(* IEC 61131-3 sources: ax-lightloop/src, 7 files *)

(* ---- LedStructs.st ---- *)
TYPE
    ///LedHw relative struct for IO assignment
    LedHw : STRUCT
        Red AT %X0.0 : BOOL;
        Yellow AT %X0.1 : BOOL;
        Green AT %X0.2 : BOOL;
    END_STRUCT;
END_TYPE

TYPE
    ///Leds array for passing bools
    Leds : STRUCT
        Red  : BOOL;
        Yellow  : BOOL;
        Green  : BOOL;
    END_STRUCT;
END_TYPE

(* ---- ILed.st ---- *)
/// Iled interface, every LED class should atleast have these functions
INTERFACE ILed
    /// GetState
    /// Method to get the state
    /// Return value: BOOL
    METHOD GetState : BOOL
    END_METHOD
    /// TurnOn
    /// Method to turn ON the LED
    /// Return value: BOOL
    METHOD TurnOn
    END_METHOD
    /// TurnOff
    /// Method to turn OFF the LED
    /// Return value: BOOL
    METHOD TurnOff
    END_METHOD

END_INTERFACE

(* ---- ITrafficLight.st ---- *)
INTERFACE ITrafficlight //ITrafficlight interfaces defines the minimum requirements for a lightstack

    /// GetState
    /// Method to get the current state of the TrafficLight
    /// Return value: state int
    METHOD GetState : int
    END_METHOD
    /// GetLedEquipmentState
    /// Method to get the current state of the Led's
    /// Return value: redHw :BOOL; yellowHw :BOOL; greenHw :BOOL;
    METHOD GetLedEquipmentState
        VAR_OUTPUT
            Leds: leds;
        END_VAR
        END_METHOD
    /// Go
    /// Method set the current state of the TrafficLight to Go
    /// Return value: success bool
    METHOD Go : BOOL
    END_METHOD
    /// Stop
    /// Method set the current state of the TrafficLight to Stop
    /// Return value: success bool
    METHOD Stop : BOOL
    END_METHOD
    /// Flash
    /// Method set the current state of the TrafficLight to Flash for idlemode
    /// Return value: none
    METHOD Flash
    END_METHOD
    /// Stop
    /// Method set the current state of the TrafficLight to Idle
    /// Return value: none
    METHOD  SetIdleMode
        VAR_INPUT
            Set : BOOL;
        END_VAR
    END_METHOD
END_INTERFACE

(* ---- led.st ---- *)
CLASS Led IMPLEMENTS Iled //This Class implements the Iled interface, to make sure it complies
    VAR PRIVATE //Private VAR section, only accesible from inside this class
        IsOn : BOOL; //Private BOOl to keep track of the LED state
    END_VAR
    ///This overwrites the comment defined in the interface
    METHOD PUBLIC GetState : BOOL
        GetState := IsOn; //Get the private state BOOL
        ;
    END_METHOD

    METHOD PUBLIC TurnOn
        IsOn := TRUE; //Set the state to ON
        ;
    END_METHOD

    METHOD PUBLIC TurnOff
        IsOn := FALSE; //Set the state to OFF
        ;
    END_METHOD

    /// Toggle
    /// This Method will Toggle the LED, this is not defined in the interface
    /// Return value: BOOL
    METHOD PUBLIC Toggle
        IF IsOn THEN //If the LED IsOn = true then set the LED to OFF
            IsOn := FALSE;
        ELSE
            IsOn := TRUE; //If the LED IsOn = false then set the LED to ON
        END_IF;
        ;
    END_METHOD

END_CLASS

(* ---- TrafficLight.st ---- *)
USING System.Timer;
CLASS Trafficlight IMPLEMENTS ITrafficlight
    VAR
        //Initialize Led classes
        Red : Led;
        Yellow : Led;
        Green : Led;

        IdleMode: BOOL := false; //Init IdleMode to false

        //Set the time that the light should be on
        YellowTime : TIME := TIME#1s;
        RedTime : TIME := TIME#1s;
        GreenTime : TIME := TIME#1s;

        Timer : System.Timer.OnDelay;
    END_VAR
    VAR PRIVATE
        state : INT; //Make sure that state cannot be manupulated from outside the class
    END_VAR

    METHOD PUBLIC GetState : Int
        GetState := state;
        ;
    END_METHOD

    METHOD PUBLIC Cycle
        VAR_INPUT

        END_VAR
        CASE State OF
            0:
                //Blink the yellow light if idlemode is active
                IF IdleMode THEN
                THIS.Flash();
                ELSE
                    Yellow.TurnOff();
                    State := 1;
                END_IF;
            1:
                //Red

                Timer(signal := NOT Timer.output, duration := RedTime);
                IF Timer.output THEN
                    Red.TurnOff();
                    Green.TurnOn();
                    State := 2;
                END_IF;
            2:
                //Green

                Timer(signal := NOT Timer.output, duration := GreenTime);
                IF Timer.output THEN
                    Green.TurnOff();
                    Yellow.TurnOn();
                    State := 3;
                END_IF;
            3:
                //Yellow

                Timer(signal := NOT Timer.output, duration := YellowTime);
                IF Timer.output THEN
                    Yellow.TurnOff();
                    Red.TurnOn();
                    State := 1;
                END_IF;
        END_CASE;
        ;
    END_METHOD

            /// Get the state of the invidual LED's
    METHOD PUBLIC GetLedEquipmentState

        VAR_OUTPUT
            Leds : Leds;
        END_VAR;
        Leds.Red := Red.GetState();
        Leds.Yellow := Yellow.GetState();
        Leds.Green := Green.GetState();
    END_METHOD

            /// Set Time for yellow light
    METHOD PUBLIC setTimeYellow

        VAR_INPUT
            DelayTime : TIME;
        END_VAR
        YellowTime := DelayTime;
        ;
    END_METHOD
///transition from red to green
    METHOD PUBLIC Go : BOOL

        IF Red.GetState() AND Yellow.GetState() = FALSE OR IdleMode THEN
            IdleMode := FALSE;
            Red.TurnOff();
            Yellow.TurnOff();
            Green.TurnOn();
            Go := TRUE;
        // ELSIF Green.GetState() = FALSE THEN
        //     THIS.SetIdleMode(true);
        END_IF;
        ;
    END_METHOD

    /// Transition from Green to Red
    METHOD PUBLIC Stop :BOOL

        IF Green.GetState() AND Yellow.GetState() = FALSE OR IdleMode OR Yellow.GetState() THEN
            Yellow.TurnOn();
            Green.TurnOff();
                Timer(signal := NOT Timer.output, duration := YellowTime);
                IF Timer.output THEN
                    // Code to turn on the light
                    IdleMode := FALSE;
                    Red.TurnOn();
                    Yellow.TurnOff();
                    Stop := TRUE;
                    ;
                END_IF;
        // ELSIF Red.GetState() = false THEN
        //     THIS.SetIdleMode(true);
        END_IF;

    END_METHOD

    METHOD PUBLIC SetIdleMode
        VAR_INPUT
            Set : BOOL;
        END_VAR
        IdleMode := Set;
        ;
    END_METHOD

    METHOD PUBLIC Flash

        //todo this should start flashing
        Timer(signal := NOT Timer.output, duration := TIME#1s);
        IF Timer.output THEN
            // Code to turn on the light
            Red.TurnOff();
            Yellow.TurnOn();
            Green.TurnOff();
            ;
        ELSE
            // Code to turn off the light
            Red.TurnOff();
            Yellow.TurnOff();
            Green.TurnOff();
            ;
        END_IF;
        ;

    END_METHOD
END_CLASS

(* ---- configuration.st ---- *)
CONFIGURATION PLC_1
    TASK Main(Interval := T#10ms, Priority := 1);
    PROGRAM P1 WITH Main: StatusLedCtrl;

    VAR_GLOBAL
        //Map LED's to HW output
        LedHw AT %QB0 : LedHw;
        //Init Trafficlight
        trafficlight : Trafficlight;
        //Some Bools to control
        idle: BOOL;
        count : INT;
    END_VAR
END_CONFIGURATION

(* ---- program.st ---- *)
PROGRAM StatusLedCtrl
    VAR_EXTERNAL
        LedHW : LedHw;
        TrafficLight : Trafficlight;
        Idle: BOOL;
        count : INT;
    END_VAR
    VAR
        SWLeds : leds;
    END_VAR

    count := count+1;
    //Get the state of the traffic light
    TrafficLight.GetLedEquipmentState(SWLeds);

    LedHW.Green := SWLeds.Green;
    LedHW.Yellow := SWLeds.Yellow;
    LedHW.Red := SWLeds.Red;

    //Execute the trafficlight statemachine
    TrafficLight.Cycle();

    //Set the trafficlight to idle if idle bool is triggered
    TrafficLight.SetIdleMode(Idle);
    ;
END_PROGRAM
